// TwinCAT 3 PLC project ProcessControl
// ProgramVersion: 3.1.4023.0
// libraries:
//   CmpBitmapPool, * (System)
//   Tc2_Standard, * (Beckhoff Automation GmbH)
//   Tc2_System, * (Beckhoff Automation GmbH)
//   Tc3_Module, * (Beckhoff Automation GmbH)
//   VisuSymbols,3.5.10.0,System
// project tree:
//   DUTs/ ATV_Status.TcDUT
//   / GlobalTextList.TcGTLO, PlcTask.TcTTO, Visualization Manager.TcVMO (not stored), VISU_TASK.TcTTO
//   GVLs/ drive.TcGVL, Pyrotime.TcGVL, Pyrotime_1.TcGVL
//   POUs/ CabinetSwitch.TcPOU, MAIN.TcPOU, FullProcess.TcPOU, FeedMotor1Manualcontrol.TcPOU, FeedMotor2Manualcontrol.TcPOU, ProcessLamp.TcPOU, RemovalProgram.TcPOU, Scaling.TcPOU, ShortProcess.TcPOU, ValveManualControl.TcPOU
//   VISUs/ ImagePool.TcIPO (not stored), Visualization.TcVIS
// real-time tasks:
//   TASK PlcTask: cycle T#10ms, priority 20, ADS port 350
//   TASK VISU_TASK: cycle T#200000us, priority 30, ADS port 351
// I/O:
//   DEVICE Device 3 (EtherCAT), AmsNetId 5.27.137.92.4.1
//     Box 2 (ATV320 EtherCAT) [ATV320 EtherCAT]
//   DEVICE Device 2 (CX-BK)
//     Box 1 (CX-BK)
// variable links:
//   ProcessControl/ProcessControl Instance <-> Device 2 (CX-BK)/Box 1 (CX-BK)
//     PlcTask Inputs/drive.RawThermoCouple1Value <-> Term 8 (KL3052)/Channel 1/Data In
//     PlcTask Inputs/drive.RawThermoCouple2Value <-> Term 8 (KL3052)/Channel 2/Data In
//     PlcTask Inputs/drive.RemovalSwitch <-> Term 2 (KL1104)/Channel 2/Input
//     PlcTask Inputs/drive.ValveSwitch <-> Term 2 (KL1104)/Channel 3/Input
//     PlcTask Inputs/drive.bEstop <-> Term 2 (KL1104)/Channel 1/Input
//     PlcTask Inputs/drive.bM1switch <-> Term 6 (KL1408)/Channel 2/Input
//     PlcTask Inputs/drive.bM2switch <-> Term 6 (KL1408)/Channel 1/Input
//     PlcTask Inputs/drive.bShortFeed <-> Term 6 (KL1408)/Channel 4/Input
//     PlcTask Inputs/drive.bStartProcess <-> Term 6 (KL1408)/Channel 3/Input
//     PlcTask Outputs/drive.CloseBottomValve <-> Term 3 (KL2114)/Channel 1/Output
//     PlcTask Outputs/drive.CloseTopValve <-> Term 3 (KL2114)/Channel 3/Output
//     PlcTask Outputs/drive.OpenBottomValve <-> Term 3 (KL2114)/Channel 4/Output
//     PlcTask Outputs/drive.OpenTopValve <-> Term 3 (KL2114)/Channel 2/Output
//     PlcTask Outputs/drive.bEmergencyLamp1 <-> Term 7 (KL2408)/Channel 3/Output
//     PlcTask Outputs/drive.bEmptySystemSwitchLamp <-> Term 5 (KL2114)/Channel 4/Output
//     PlcTask Outputs/drive.bFeedMotor2 <-> Term 7 (KL2408)/Channel 6/Output
//     PlcTask Outputs/drive.bM1active <-> Term 4 (KL2114)/Channel 4/Output
//     PlcTask Outputs/drive.bM2active <-> Term 4 (KL2114)/Channel 3/Output
//     PlcTask Outputs/drive.bProcessActive <-> Term 4 (KL2114)/Channel 1/Output
//     PlcTask Outputs/drive.bRemovalMotor <-> Term 5 (KL2114)/Channel 1/Output
//     PlcTask Outputs/drive.bRemovalSequenceLamp <-> Term 5 (KL2114)/Channel 2/Output
//     PlcTask Outputs/drive.bVacuum <-> Term 7 (KL2408)/Channel 5/Output
//     PlcTask Outputs/drive.bValveLamp <-> Term 4 (KL2114)/Channel 2/Output
//     PlcTask Outputs/drive.bValveSwitchLamp <-> Term 5 (KL2114)/Channel 3/Output
//     PlcTask Outputs/drive.bfeedmotorSwitchlamp <-> Term 7 (KL2408)/Channel 2/Output
//     PlcTask Outputs/drive.bremovalmotorSwitchlamp <-> Term 7 (KL2408)/Channel 1/Output
//     PlcTask Outputs/drive.bstartprocessSwitchlamp <-> Term 7 (KL2408)/Channel 4/Output
//   ProcessControl/ProcessControl Instance <-> Device 3 (EtherCAT)/Box 2 (ATV320 EtherCAT)
//     PlcTask Inputs/drive.ATV_TPDO_Input1_Status_Word <-> Inputs/Status word
//     PlcTask Inputs/drive.ATV_TPDO_Input2_Control_Effort <-> Inputs/Control Effort
//     PlcTask Outputs/drive.ATV_RPDO_Output1_Control_Word <-> Outputs/Control word
//     PlcTask Outputs/drive.ATV_RPDO_Output2_Target_Velocity <-> Outputs/Target Velocity

CONFIGURATION ProcessControl
    RESOURCE PLC ON TwinCAT3
        TASK PlcTask(INTERVAL := T#10ms, PRIORITY := 20);
        TASK VISU_TASK(INTERVAL := T#200000us, PRIORITY := 30);
        PROGRAM MAIN WITH PlcTask : MAIN;
        PROGRAM VisuElems_Visu_Prg WITH VISU_TASK : VisuElems.Visu_Prg;
    END_RESOURCE
END_CONFIGURATION

// ---- DUTs/ATV_Status.TcDUT
{attribute 'qualified_only'}
{attribute 'strict'}
TYPE ATV_Status :
(
    SwitchON_disabled := 592, //0
	rdy2SwitchON := 561,	// 6 
	SwitchedON := 563,		// 7 hexadecimal. Motor is in a state, ready to be turned on but not actually on
	OP_Enabled := 1591		//15 hexadecimal. Motor is actually in operation
)   WORD := SwitchON_disabled;
END_TYPE

// ---- GVLs/drive.TcGVL
{attribute 'qualified_only'}
VAR_GLOBAL
	// -------- motor 1 params --------------------------	
	ATV_State AT %I* : WORD;
	PLC_state AT %I* : UINT;
	ATV_TPDO_Input1_Status_Word AT %I* : WORD;
	ATV_TPDO_Input2_Control_Effort AT %I* : WORD;
	ATV_TPDO_Input3 AT %I* : WORD; 
	ATV_TPDO_Input4 AT %I* : WORD;
	ATV_TPDO_Input5 AT %I* : WORD;
	ATV_TPDO_Input6 AT %I* : WORD;
	ATV_RPDO_Output1_Control_Word AT %Q* : WORD;
	ATV_RPDO_Output2_Target_Velocity AT %Q* : WORD;
	ATV_RPDO_Output3 AT %Q* : WORD; 
	ATV_RPDO_Output4 AT %Q* : WORD; 
	ATV_RPDO_Output5 AT %Q* : WORD; 
	ATV_RPDO_Output6 AT %Q* : WORD; 
// -------- motor 1 params --------------------------

// -------- motor 2 params --------------------------
{attribute 'OPC.UA.DA' := '1'} 
bRemovalMotor AT %Q* : BOOL;
// -------- motor 2 params --------------------------

//------------ fan params ----------------
{attribute 'OPC.UA.DA' := '1'} 
bGasfan AT %Q* : BOOL;
//------------- fan params ------------------

//---------- motor 3 params--------------------------
{attribute 'OPC.UA.DA' := '1'} 
bFeedMotor2 AT %Q* : BOOL;
//----------- motor 3 params ------------------------

//---------- switches -------------------------------
{attribute 'OPC.UA.DA' := '1'} 
bStartProcess AT %I* :BOOL;

bEstop      AT %I* 	 :BOOL; 

bM1switch AT %I* 	 :BOOL; 

bM2switch AT %I* 	 :BOOL;

RemovalSwitch AT %I* :BOOL;

{attribute 'OPC.UA.DA' := '1'} 
bShortFeed AT %I* 	 :BOOL; 

bCompressor  	 	 :BOOL; 

{attribute 'OPC.UA.DA' := '1'} 
ValveSwitch AT %I* 	 :BOOL;
//---------- switches -----------------------------

// ---------Lamps----------------------------------
// lamps on the door of the cabinet 
bEmergencyLamp1 AT %Q*   :BOOL; 

{attribute 'OPC.UA.DA' := '1'} 
bProcessActive AT %Q*    :BOOL;
 
bRemovalSequenceLamp AT %Q*   :BOOL;

{attribute 'OPC.UA.DA' := '1'} 
bM1active 		AT %Q* 	 :BOOL;

{attribute 'OPC.UA.DA' := '1'} 
bM2active		AT %Q* 	 :BOOL;

bVacuumActive   AT %Q* 	 :BOOL; 

bValveLamp AT %Q* 		 :BOOL; 

bFeedMotor2Lamp AT %Q*   :BOOL;

//----- lamps inside the switches -------------
bstartprocessSwitchlamp AT %Q* :BOOL;

bfeedmotorSwitchlamp AT %Q* :BOOL; 

bremovalmotorSwitchlamp AT %Q* :BOOL;  

bValveSwitchLamp AT %Q* :BOOL;

bEmptySystemSwitchLamp at %Q* :BOOL; 
// ---------Lamps-----------------------------------

//----------- counter variables ---------------------

ifeedmotor1count: INT;
itopvalvecount: INT := 1;

//----------- counter variables ---------------------


//----status variables-------------
bM1run  	 :BOOL;
ProcessActive :BOOL;
bM1status    : BOOL;    				// tells if the motor is on/off
//-----status variables------------



//---------Valve control ------------------------------------
{attribute 'OPC.UA.DA' := '1'} 
OpenTopValve AT %Q* : BOOL;

{attribute 'OPC.UA.DA' := '1'} 
CloseTopValve AT %Q*: BOOL;
 
{attribute 'OPC.UA.DA' := '1'} 
OpenBottomValve AT %Q* : BOOL;

{attribute 'OPC.UA.DA' := '1'} 
CloseBottomValve AT %Q*: BOOL; 
//----------Valve control -----------------------------------

//----- Vacuum pump --------------------------------------
{attribute 'OPC.UA.DA' := '1'} 
bVacuum  AT %Q*	 : BOOL;
//-----Vacuum pump ---------------------------------------


//------------Temperature variables ---------------------------
RawThermoCouple1Value  AT %I* :INT;
ScaledThermoCouple1Value: REAL; 
RawThermoCouple2Value AT %I*: INT;

{attribute 'OPC.UA.DA' := '1'} 
ScaledThermoCouple2Value: REAL; 
//-----------Temperature variables -----------------------------

END_VAR

// ---- GVLs/Pyrotime.TcGVL
{attribute 'qualified_only'}

// Times used for testing.
VAR_GLOBAL
	tStartDelay: TIME := T#1S;
	tInitFeed: TIME := T#344S; //344s
	tShortFeed: TIME := T#118S; //118s
	tTempFall: TIME:= T#2S;
	tRemovalMotor: TIME := T#114S; //114s
	tValve2: TIME := T#3S;
	tVacuum: TIME := t#10s;
END_VAR

// ---- GVLs/Pyrotime_1.TcGVL
{attribute 'qualified_only'}

// These times are for testing. They are much shorter than the original times
VAR_GLOBAL
	tStartDelay: TIME := T#1S;
	tInitFeed: TIME := T#4S; //344s
	tShortFeed: TIME := T#5S; //118s
	tTempFall: TIME:= T#2S;
	tRemovalMotor: TIME := T#5S; //114s
	tValve2: TIME := T#2S;
END_VAR

// ---- POUs/MAIN.TcPOU
PROGRAM MAIN
VAR
END_VAR

ProcessLamp();
FullProcess();
ShortProcess(); 
FeedMotor1Manualcontrol();
CabinetSwitch();
ValveManualControl();
Scaling();
FeedMotor2Manualcontrol();
RemovalProgram();

END_PROGRAM

// ---- POUs/ProcessLamp.TcPOU
PROGRAM ProcessLamp
VAR
END_VAR

// Written 10.08.2023 by Daniel Kelly

// The purpose of this POU is to provide control to the lamps on the 
// front of the cabinet via their switches

drive.bM1active := drive.bM1switch;
drive.bM2active := drive.bM2switch; 
drive.bProcessActive := drive.bShortFeed OR drive.bStartProcess;
drive.bRemovalSequenceLamp := drive.RemovalSwitch;
drive.bValveLamp := drive.ValveSwitch;

END_PROGRAM

// ---- POUs/FullProcess.TcPOU
PROGRAM FullProcess
VAR
END_VAR
// written 7.08.2023 by Daniel Kelly

// This program is the full version of the process. It includes longer feeding 
// and residence times
// RValveOff turns off the solenoids on the righthandside incase they were already on
// OpenValve opens the top valve
// Step Vacuum removes the excess air from inside the pipe via the vacuum
//waitTemp waits until the temperature is at least 350 degrees celsius
// BiomassFeed operates the second feeding motor
// Init_Feed operates the main feeding motor
// wait600 waits until temperature is 600
// GasFanON turns on the gas fan
// ShortFeed turns on the main feeding motor 1
// ExitMotor turns on the removal motor and opens the top valve
// Valve2Open opens the bottom valve
// Valve2Close closes the bottom valve
// SolenoidsOff turns off the solenoids incase they were on
// AirRemoval removes the air from the pipe
// turnoff1 etc. turns off the devices such as the valves and feeding motor 2

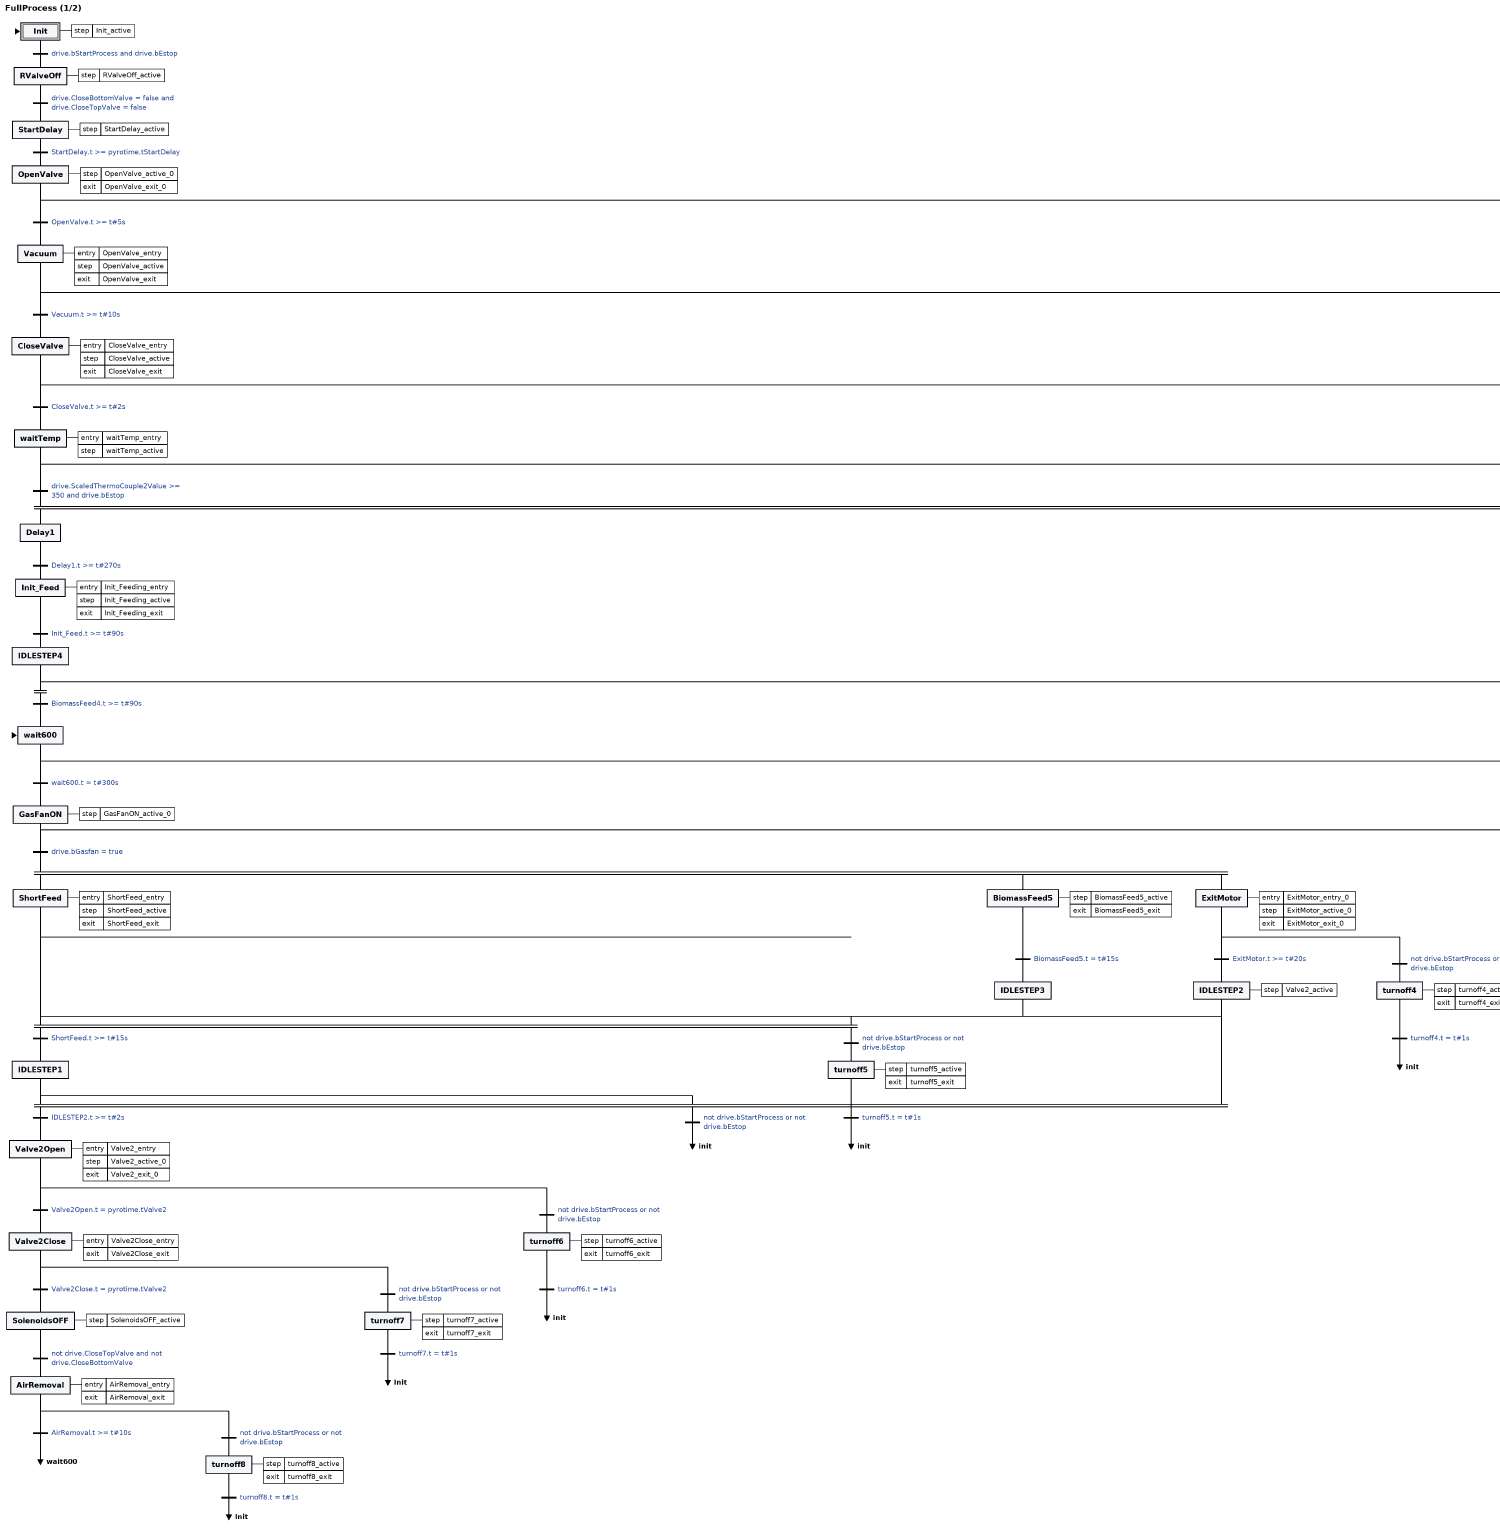
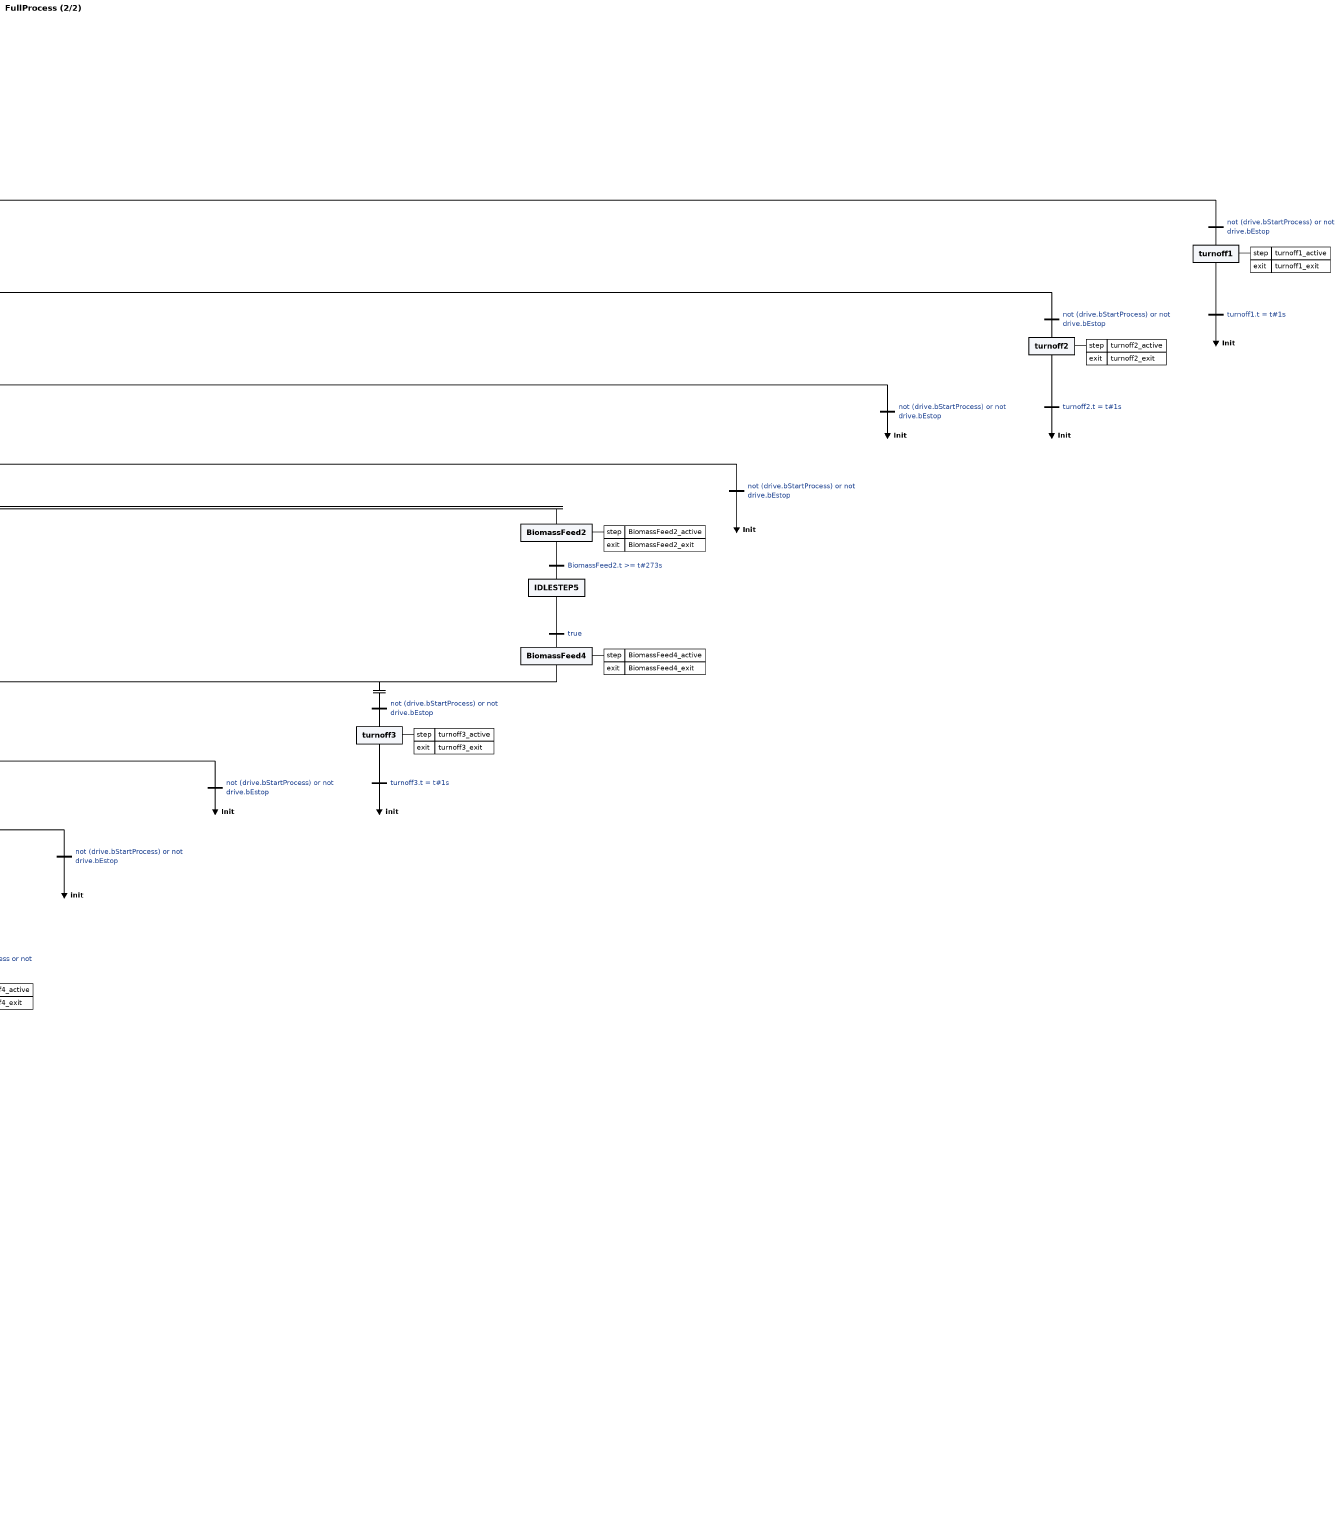
INITIAL_STEP Init:
    Init_active(N);  // step action
END_STEP
TRANSITION FROM Init TO RValveOff
    := drive.bStartProcess and drive.bEstop;
END_TRANSITION
STEP RValveOff:
    RValveOff_active(N);  // step action
END_STEP
TRANSITION FROM RValveOff TO StartDelay
    := drive.CloseBottomValve = false and drive.CloseTopValve = false;
END_TRANSITION
STEP StartDelay:
    StartDelay_active(N);  // step action
END_STEP
TRANSITION FROM StartDelay TO OpenValve
    := StartDelay.t >= pyrotime.tStartDelay;
END_TRANSITION
STEP OpenValve:
    OpenValve_active_0(N);  // step action
    OpenValve_exit_0(P0);  // exit action
END_STEP
TRANSITION FROM OpenValve TO Vacuum
    := OpenValve.t >= t#5s;
END_TRANSITION
TRANSITION FROM OpenValve TO turnoff1
    := not (drive.bStartProcess) or not drive.bEstop;
END_TRANSITION
STEP turnoff1:
    turnoff1_active(N);  // step action
    turnoff1_exit(P0);  // exit action
END_STEP
TRANSITION FROM turnoff1 TO Init
    := turnoff1.t = t#1s;
END_TRANSITION
STEP Vacuum:
    OpenValve_entry(P1);  // entry action
    OpenValve_active(N);  // step action
    OpenValve_exit(P0);  // exit action
END_STEP
TRANSITION FROM Vacuum TO CloseValve
    := Vacuum.t >= t#10s;
END_TRANSITION
TRANSITION FROM Vacuum TO turnoff2
    := not (drive.bStartProcess) or not drive.bEstop;
END_TRANSITION
STEP turnoff2:
    turnoff2_active(N);  // step action
    turnoff2_exit(P0);  // exit action
END_STEP
TRANSITION FROM turnoff2 TO Init
    := turnoff2.t = t#1s;
END_TRANSITION
STEP CloseValve:
    CloseValve_entry(P1);  // entry action
    CloseValve_active(N);  // step action
    CloseValve_exit(P0);  // exit action
END_STEP
TRANSITION FROM CloseValve TO waitTemp
    := CloseValve.t >= t#2s;
END_TRANSITION
TRANSITION FROM CloseValve TO Init
    := not (drive.bStartProcess) or not drive.bEstop;
END_TRANSITION
STEP waitTemp:
    waitTemp_entry(P1);  // entry action
    waitTemp_active(N);  // step action
END_STEP
TRANSITION FROM waitTemp TO (Delay1, BiomassFeed2)
    := drive.ScaledThermoCouple2Value >= 350 and drive.bEstop;
END_TRANSITION
TRANSITION FROM waitTemp TO Init
    := not (drive.bStartProcess) or not drive.bEstop;
END_TRANSITION
STEP Delay1:
END_STEP
TRANSITION FROM Delay1 TO Init_Feed
    := Delay1.t >= t#270s;
END_TRANSITION
STEP Init_Feed:
    Init_Feeding_entry(P1);  // entry action
    Init_Feeding_active(N);  // step action
    Init_Feeding_exit(P0);  // exit action
END_STEP
TRANSITION FROM Init_Feed TO IDLESTEP4
    := Init_Feed.t >= t#90s;
END_TRANSITION
STEP IDLESTEP4:
END_STEP
STEP BiomassFeed2:
    BiomassFeed2_active(N);  // step action
    BiomassFeed2_exit(P0);  // exit action
END_STEP
TRANSITION FROM BiomassFeed2 TO IDLESTEP5
    := BiomassFeed2.t >= t#273s;
END_TRANSITION
STEP IDLESTEP5:
END_STEP
TRANSITION FROM IDLESTEP5 TO BiomassFeed4
    := true;
END_TRANSITION
STEP BiomassFeed4:
    BiomassFeed4_active(N);  // step action
    BiomassFeed4_exit(P0);  // exit action
END_STEP
TRANSITION FROM (IDLESTEP4, BiomassFeed4) TO wait600
    := BiomassFeed4.t >= t#90s;
END_TRANSITION
TRANSITION FROM (IDLESTEP4, BiomassFeed4) TO turnoff3
    := not (drive.bStartProcess) or not drive.bEstop;
END_TRANSITION
STEP turnoff3:
    turnoff3_active(N);  // step action
    turnoff3_exit(P0);  // exit action
END_STEP
TRANSITION FROM turnoff3 TO init
    := turnoff3.t = t#1s;
END_TRANSITION
STEP wait600:
END_STEP
TRANSITION FROM wait600 TO GasFanON
    := wait600.t = t#300s;
END_TRANSITION
STEP GasFanON:
    GasFanON_active_0(N);  // step action
END_STEP
TRANSITION FROM GasFanON TO (ShortFeed, BiomassFeed5, ExitMotor)
    := drive.bGasfan = true;
END_TRANSITION
TRANSITION FROM GasFanON TO init
    := not (drive.bStartProcess) or not drive.bEstop;
END_TRANSITION
TRANSITION FROM wait600 TO Init
    := not (drive.bStartProcess) or not drive.bEstop;
END_TRANSITION
STEP ShortFeed:
    ShortFeed_entry(P1);  // entry action
    ShortFeed_active(N);  // step action
    ShortFeed_exit(P0);  // exit action
END_STEP
STEP BiomassFeed5:
    BiomassFeed5_active(N);  // step action
    BiomassFeed5_exit(P0);  // exit action
END_STEP
TRANSITION FROM BiomassFeed5 TO IDLESTEP3
    := BiomassFeed5.t = t#15s;
END_TRANSITION
STEP IDLESTEP3:
END_STEP
TRANSITION FROM (ShortFeed, IDLESTEP3) TO IDLESTEP1
    := ShortFeed.t >= t#15s;
END_TRANSITION
TRANSITION FROM (ShortFeed, IDLESTEP3) TO turnoff5
    := not drive.bStartProcess or not drive.bEstop;
END_TRANSITION
STEP turnoff5:
    turnoff5_active(N);  // step action
    turnoff5_exit(P0);  // exit action
END_STEP
TRANSITION FROM turnoff5 TO init
    := turnoff5.t = t#1s;
END_TRANSITION
STEP IDLESTEP1:
END_STEP
STEP ExitMotor:
    ExitMotor_entry_0(P1);  // entry action
    ExitMotor_active_0(N);  // step action
    ExitMotor_exit_0(P0);  // exit action
END_STEP
TRANSITION FROM ExitMotor TO IDLESTEP2
    := ExitMotor.t >= t#20s;
END_TRANSITION
TRANSITION FROM ExitMotor TO turnoff4
    := not drive.bStartProcess or not drive.bEstop;
END_TRANSITION
STEP turnoff4:
    turnoff4_active(N);  // step action
    turnoff4_exit(P0);  // exit action
END_STEP
TRANSITION FROM turnoff4 TO init
    := turnoff4.t = t#1s;
END_TRANSITION
STEP IDLESTEP2:
    Valve2_active(N);  // step action
END_STEP
TRANSITION FROM (IDLESTEP1, IDLESTEP2) TO Valve2Open
    := IDLESTEP2.t >= t#2s;
END_TRANSITION
TRANSITION FROM (IDLESTEP1, IDLESTEP2) TO init
    := not drive.bStartProcess or not drive.bEstop;
END_TRANSITION
STEP Valve2Open:
    Valve2_entry(P1);  // entry action
    Valve2_active_0(N);  // step action
    Valve2_exit_0(P0);  // exit action
END_STEP
TRANSITION FROM Valve2Open TO Valve2Close
    := Valve2Open.t = pyrotime.tValve2;
END_TRANSITION
TRANSITION FROM Valve2Open TO turnoff6
    := not drive.bStartProcess or not drive.bEstop;
END_TRANSITION
STEP turnoff6:
    turnoff6_active(N);  // step action
    turnoff6_exit(P0);  // exit action
END_STEP
TRANSITION FROM turnoff6 TO init
    := turnoff6.t = t#1s;
END_TRANSITION
STEP Valve2Close:
    Valve2Close_entry(P1);  // entry action
    Valve2Close_exit(P0);  // exit action
END_STEP
TRANSITION FROM Valve2Close TO SolenoidsOFF
    := Valve2Close.t = pyrotime.tValve2;
END_TRANSITION
TRANSITION FROM Valve2Close TO turnoff7
    := not drive.bStartProcess or not drive.bEstop;
END_TRANSITION
STEP turnoff7:
    turnoff7_active(N);  // step action
    turnoff7_exit(P0);  // exit action
END_STEP
TRANSITION FROM turnoff7 TO Init
    := turnoff7.t = t#1s;
END_TRANSITION
STEP SolenoidsOFF:
    SolenoidsOFF_active(N);  // step action
END_STEP
TRANSITION FROM SolenoidsOFF TO AirRemoval
    := not drive.CloseTopValve and not drive.CloseBottomValve;
END_TRANSITION
STEP AirRemoval:
    AirRemoval_entry(P1);  // entry action
    AirRemoval_exit(P0);  // exit action
END_STEP
TRANSITION FROM AirRemoval TO wait600
    := AirRemoval.t >= t#10s;
END_TRANSITION
TRANSITION FROM AirRemoval TO turnoff8
    := not drive.bStartProcess or not drive.bEstop;
END_TRANSITION
STEP turnoff8:
    turnoff8_active(N);  // step action
    turnoff8_exit(P0);  // exit action
END_STEP
TRANSITION FROM turnoff8 TO Init
    := turnoff8.t = t#1s;
END_TRANSITION

ACTION AirRemoval_entry:
drive.bVacuum := TRUE;
END_ACTION

ACTION AirRemoval_exit:
drive.bVacuum := FALSE;
END_ACTION

ACTION BiomassFeed_active:
drive.bFeedMotor2 := true;
END_ACTION

ACTION BiomassFeed_exit:
drive.bFeedMotor2 := false;
END_ACTION

ACTION BiomassFeed2_active:
drive.bFeedMotor2 := TRUE;
END_ACTION

ACTION BiomassFeed2_exit:
drive.bFeedMotor2 := FALSE;
END_ACTION

ACTION BiomassFeed4_active:
drive.bFeedMotor2 := TRUE;
END_ACTION

ACTION BiomassFeed4_exit:
drive.bFeedMotor2 := false;
END_ACTION

ACTION BiomassFeed5_active:
drive.bFeedMotor2 := true;
END_ACTION

ACTION BiomassFeed5_exit:
drive.bFeedMotor2 := false;
END_ACTION

ACTION CloseValve_active:
drive.CloseTopValve := TRUE;
drive.CloseBottomValve := FALSE;
END_ACTION

ACTION CloseValve_entry:
//drive.RightSolenoid := TRUE;
END_ACTION

ACTION CloseValve_exit:
drive.CloseTopValve := FALSE;
END_ACTION

ACTION ExitMotor_active_0:
drive.bRemovalMotor := TRUE;
drive.bM2active := TRUE; // lamp variable



drive.OpenTopValve := TRUE; // opens valve
drive.CloseTopValve := FALSE;
END_ACTION

ACTION ExitMotor_entry_0:

END_ACTION

ACTION ExitMotor_exit_0:
 
drive.CloseTopValve := TRUE; //closes valve
drive.OpenTopValve := FALSE;

drive.bM2active := FALSE; // lamp variable ; turns lamp off
drive.bRemovalMotor := FALSE; // turns the removal motor off
END_ACTION

ACTION ExitMotor1_active:
drive.bRemovalMotor := TRUE;
END_ACTION

ACTION GasFanOFF_active:
drive.bGasfan := false;
END_ACTION

ACTION GasFanOFF_active_0:
drive.bGasfan := false;
END_ACTION

ACTION GasFanOn_active:
drive.bGasfan := TRUE;
END_ACTION

ACTION GasFanON_active_0:
drive.bGasfan := TRUE;
END_ACTION

ACTION Init_active:
//drive.ATV_RPDO_Output1_Control_Word := 0;
//drive.bRemovalMotor := FALSE; 
//drive.bProcessActive := FALSE;
//drive.LeftSolenoid := FALSE;
//drive.LeftSolenoid2 := FALSE; 
//drive.RightSolenoid := TRUE;
//drive.RightSolenoid2 := TRUE;
 
drive.ifeedmotor1count := 0;
END_ACTION

ACTION Init_Feeding_active:
IF drive.ATV_TPDO_Input1_Status_Word = ATV_Status.rdy2SwitchON THEN 
	drive.ATV_RPDO_Output1_Control_Word := 7; //SwitchedON
END_IF

IF drive.ATV_TPDO_Input1_Status_Word = ATV_Status.SwitchedON THEN 
	drive.ATV_RPDO_Output1_Control_Word := 15; //OP_Enabled
	drive.bM1active := TRUE; // lamp goes on
	drive.bM1status := TRUE;  // status variable
END_IF
END_ACTION

ACTION Init_Feeding_entry:
drive.ATV_RPDO_Output1_Control_Word := 6; //rdy2SwitchON
drive.ATV_RPDO_Output2_Target_Velocity := 1000;
END_ACTION

ACTION Init_Feeding_exit:


IF drive.bM1status = TRUE THEN 
	drive.ifeedmotor1count := drive.ifeedmotor1count + 1;
END_IF

drive.ATV_RPDO_Output1_Control_Word := 7; //switchedON, ready mode
drive.bM1active := FALSE;  // lamp off
drive.bM1status := FALSE;  // status variable for feeding motor 1
END_ACTION

ACTION OpenValve_active:

END_ACTION

ACTION OpenValve_active_0:
drive.OpenTopValve := TRUE;
drive.CloseTopValve := FALSE;
END_ACTION

ACTION OpenValve_entry:

drive.bVacuum := TRUE;
END_ACTION

ACTION OpenValve_exit:
drive.bVacuum := FALSE;
END_ACTION

ACTION OpenValve_exit_0:
drive.OpenTopValve := false;
END_ACTION

ACTION ProcessActive_active:
IF drive.bStartProcess THEN 
	drive.bProcessActive := TRUE;
ELSE 
	drive.bProcessActive := FALSE; 
END_IF
END_ACTION

ACTION RValveOff_active:
drive.CloseTopValve := FALSE;
drive.CloseBottomValve := FALSE;
END_ACTION

ACTION ShortFeed_active:
IF drive.ATV_TPDO_Input1_Status_Word = ATV_Status.rdy2SwitchON THEN 
	drive.ATV_RPDO_Output1_Control_Word := 7;
END_IF

IF drive.ATV_TPDO_Input1_Status_Word = ATV_Status.SwitchedON THEN
			drive.bM1run := TRUE; //counter variable
			drive.bM1active := TRUE;
			drive.ATV_RPDO_Output1_Control_Word := 15;
END_IF
END_ACTION

ACTION ShortFeed_entry:
drive.ATV_RPDO_Output2_Target_Velocity := 1000;
drive.ATV_RPDO_Output1_Control_Word := 6;
END_ACTION

ACTION ShortFeed_exit:


drive.bM1run := FALSE;
drive.bM1active := FALSE; 
drive.ATV_RPDO_Output1_Control_Word := 7;
END_ACTION

ACTION SolenoidsOFF_active:
drive.CloseTopValve := FALSE;
drive.CloseBottomValve := FALSE;
END_ACTION

ACTION StartDelay_active:
IF drive.bStartProcess THEN 
	drive.bProcessActive := TRUE;
ELSE 
	drive.bProcessActive := FALSE; 
END_IF
END_ACTION

ACTION turnoff1_active:
drive.CloseTopValve := TRUE;
drive.OpenTopValve := FALSE;
END_ACTION

ACTION turnoff1_exit:
drive.CloseTopValve := FALSE;
END_ACTION

ACTION turnoff2_active:
drive.bVacuum := FALSE;
END_ACTION

ACTION turnoff2_exit:

END_ACTION

ACTION turnoff3_active:
drive.bM1status := FALSE;
drive.bFeedMotor2 := FALSE;
drive.bM1active := FALSE;
END_ACTION

ACTION turnoff3_exit:

END_ACTION

ACTION turnoff4_active:
drive.bRemovalMotor := FALSE;
drive.bM2active := FALSE;

drive.OpenTopValve := FALSE;
drive.CloseTopValve := TRUE;
END_ACTION

ACTION turnoff4_exit:
drive.CloseTopValve := false;
END_ACTION

ACTION turnoff5_active:
drive.bFeedMotor2 := FALSE;


drive.bRemovalMotor := FALSE;
drive.bM2active := FALSE;

drive.OpenTopValve := FALSE;
drive.CloseTopValve := TRUE;
END_ACTION

ACTION turnoff5_exit:

END_ACTION

ACTION turnoff6_active:
drive.CloseBottomValve := TRUE;
drive.OpenBottomValve := FALSE;
END_ACTION

ACTION turnoff6_exit:
drive.CloseBottomValve := FALSE;
END_ACTION

ACTION turnoff7_active:
drive.CloseBottomValve := TRUE;
END_ACTION

ACTION turnoff7_exit:
drive.CloseBottomValve := FALSE;
END_ACTION

ACTION turnoff8_active:
drive.bVacuum := false;
END_ACTION

ACTION turnoff8_exit:

END_ACTION

ACTION Vacuum_entry:

END_ACTION

ACTION Vacuum_exit:
drive.bVacuum := FALSE;
END_ACTION

ACTION Valve2_active:

END_ACTION

ACTION Valve2_active_0:

END_ACTION

ACTION Valve2_entry:
drive.OpenBottomValve := TRUE;
END_ACTION

ACTION Valve2_exit_0:
drive.OpenBottomValve := FALSE;
END_ACTION

ACTION Valve2Close_entry:
drive.CloseBottomValve := TRUE;
END_ACTION

ACTION Valve2Close_exit:
 drive.CloseBottomValve := FALSE;
END_ACTION

ACTION waitTemp_active:

END_ACTION

ACTION waitTemp_entry:

END_ACTION

END_PROGRAM

// ---- POUs/ShortProcess.TcPOU
	PROGRAM ShortProcess
VAR
	cM1startCount : INT;
	
END_VAR
// written 7.08.2023 by Daniel Kelly

// Program is a shorter version of the full process cycle

//Step RValveOff turns off the top and bottom closing valves
// Step Wait500 waits until the temperature is at 500
//Step GasFanOn turns on the gas fan
// Step waittemp is the residence time
//Step ShortFeed and Biomass Feed run simultaneously to feed the biomass into the furnace
// Step ExitMotor operates the removal motor and opens the top valve
// Steps M1override and M2override overrides the original motor operating time.
//Step Valve2Open opens the bottom valve
// Step Valve2Close closes the bottom valve

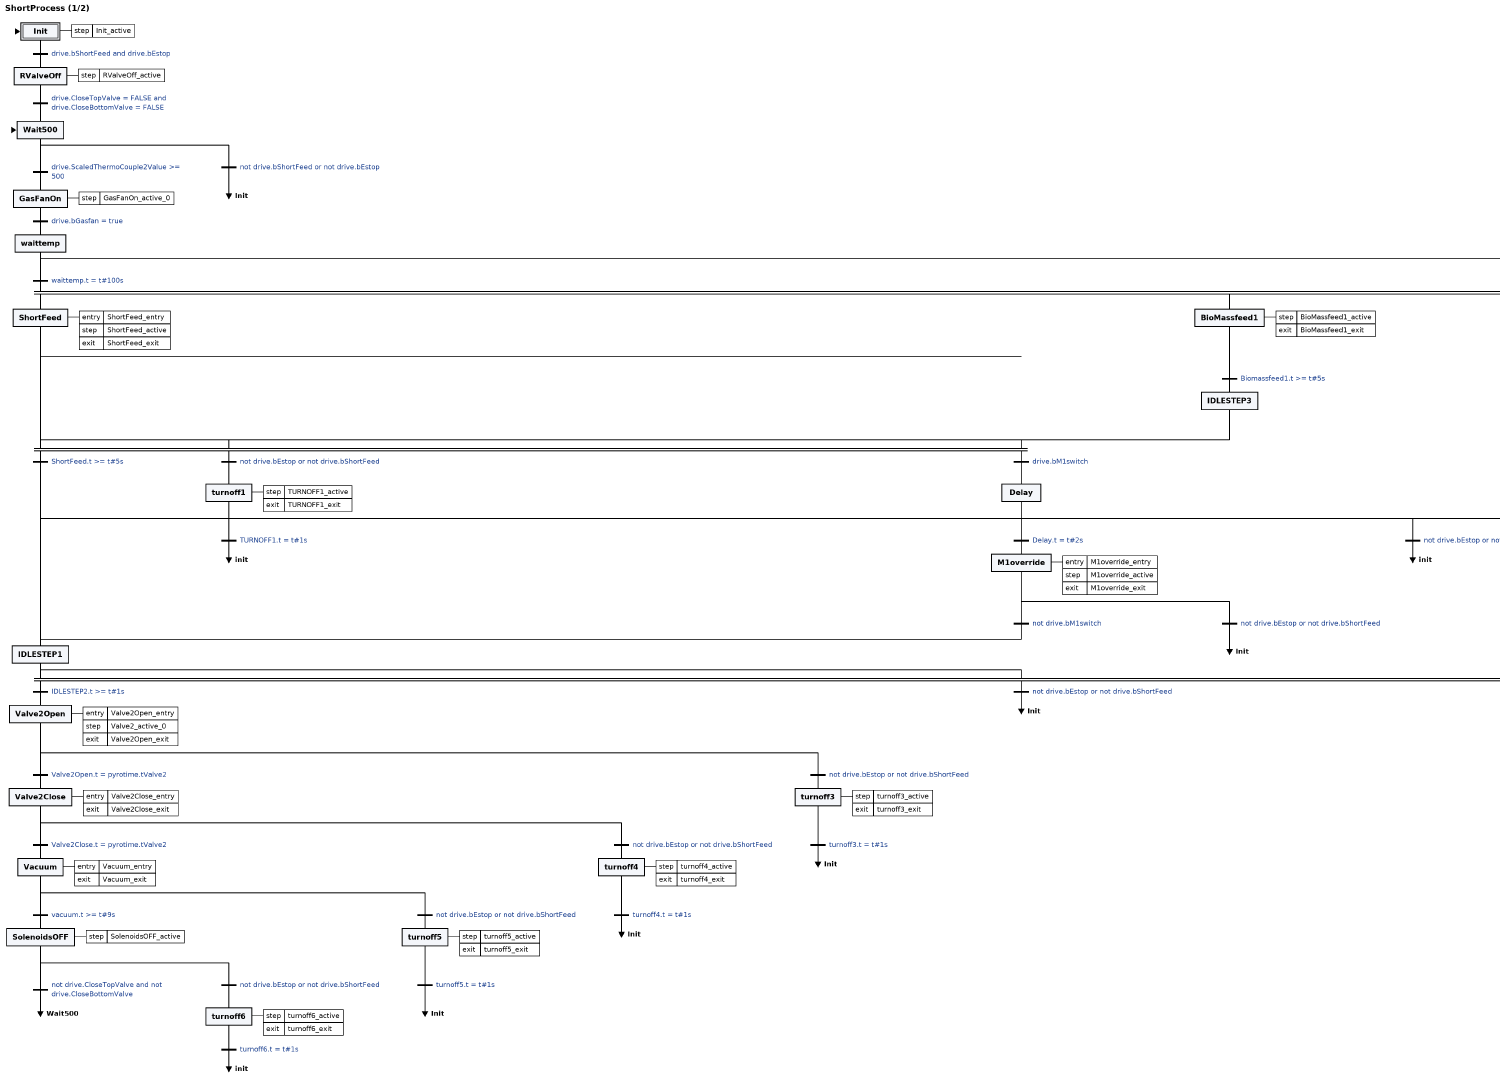
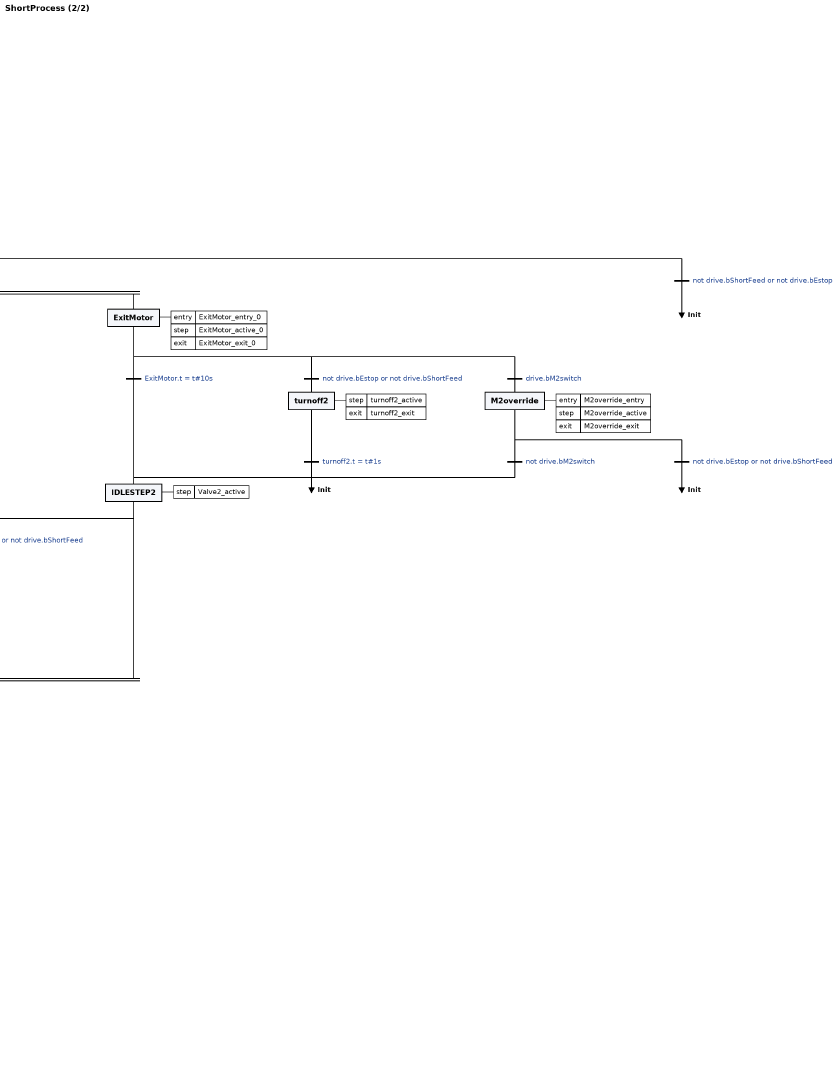
INITIAL_STEP Init:
    Init_active(N);  // step action
END_STEP
TRANSITION FROM Init TO RValveOff
    := drive.bShortFeed and drive.bEstop;
END_TRANSITION
STEP RValveOff:
    RValveOff_active(N);  // step action
END_STEP
TRANSITION FROM RValveOff TO Wait500
    := drive.CloseTopValve = FALSE and drive.CloseBottomValve = FALSE;
END_TRANSITION
STEP Wait500:
END_STEP
TRANSITION FROM Wait500 TO GasFanOn
    := drive.ScaledThermoCouple2Value >= 500;
END_TRANSITION
STEP GasFanOn:
    GasFanOn_active_0(N);  // step action
END_STEP
TRANSITION FROM GasFanOn TO waittemp
    := drive.bGasfan = true;
END_TRANSITION
TRANSITION FROM Wait500 TO Init
    := not drive.bShortFeed or not drive.bEstop;
END_TRANSITION
STEP waittemp:
END_STEP
TRANSITION FROM waittemp TO (ShortFeed, BioMassfeed1, ExitMotor)
    := waittemp.t = t#100s;
END_TRANSITION
TRANSITION FROM waittemp TO Init
    := not drive.bShortFeed or not drive.bEstop;
END_TRANSITION
STEP ShortFeed:
    ShortFeed_entry(P1);  // entry action
    ShortFeed_active(N);  // step action
    ShortFeed_exit(P0);  // exit action
END_STEP
STEP BioMassfeed1:
    BioMassfeed1_active(N);  // step action
    BioMassfeed1_exit(P0);  // exit action
END_STEP
TRANSITION FROM BioMassfeed1 TO IDLESTEP3
    := Biomassfeed1.t >= t#5s;
END_TRANSITION
STEP IDLESTEP3:
END_STEP
TRANSITION FROM (ShortFeed, IDLESTEP3) TO IDLESTEP1
    := ShortFeed.t >= t#5s;
END_TRANSITION
TRANSITION FROM (ShortFeed, IDLESTEP3) TO turnoff1
    := not drive.bEstop or not drive.bShortFeed;
END_TRANSITION
STEP turnoff1:
    TURNOFF1_active(N);  // step action
    TURNOFF1_exit(P0);  // exit action
END_STEP
TRANSITION FROM turnoff1 TO init
    := TURNOFF1.t = t#1s;
END_TRANSITION
TRANSITION FROM (ShortFeed, IDLESTEP3) TO Delay
    := drive.bM1switch;
END_TRANSITION
STEP Delay:
END_STEP
TRANSITION FROM Delay TO M1override
    := Delay.t = t#2s;
END_TRANSITION
TRANSITION FROM Delay TO init
    := not drive.bEstop or not drive.bShortFeed;
END_TRANSITION
STEP M1override:
    M1override_entry(P1);  // entry action
    M1override_active(N);  // step action
    M1override_exit(P0);  // exit action
END_STEP
TRANSITION FROM M1override TO IDLESTEP1
    := not drive.bM1switch;
END_TRANSITION
TRANSITION FROM M1override TO Init
    := not drive.bEstop or not drive.bShortFeed;
END_TRANSITION
STEP IDLESTEP1:
END_STEP
STEP ExitMotor:
    ExitMotor_entry_0(P1);  // entry action
    ExitMotor_active_0(N);  // step action
    ExitMotor_exit_0(P0);  // exit action
END_STEP
TRANSITION FROM ExitMotor TO IDLESTEP2
    := ExitMotor.t = t#10s;
END_TRANSITION
TRANSITION FROM ExitMotor TO turnoff2
    := not drive.bEstop or not drive.bShortFeed;
END_TRANSITION
STEP turnoff2:
    turnoff2_active(N);  // step action
    turnoff2_exit(P0);  // exit action
END_STEP
TRANSITION FROM turnoff2 TO Init
    := turnoff2.t = t#1s;
END_TRANSITION
TRANSITION FROM ExitMotor TO M2override
    := drive.bM2switch;
END_TRANSITION
STEP M2override:
    M2override_entry(P1);  // entry action
    M2override_active(N);  // step action
    M2override_exit(P0);  // exit action
END_STEP
TRANSITION FROM M2override TO IDLESTEP2
    := not drive.bM2switch;
END_TRANSITION
TRANSITION FROM M2override TO Init
    := not drive.bEstop or not drive.bShortFeed;
END_TRANSITION
STEP IDLESTEP2:
    Valve2_active(N);  // step action
END_STEP
TRANSITION FROM (IDLESTEP1, IDLESTEP2) TO Valve2Open
    := IDLESTEP2.t >= t#1s;
END_TRANSITION
TRANSITION FROM (IDLESTEP1, IDLESTEP2) TO Init
    := not drive.bEstop or not drive.bShortFeed;
END_TRANSITION
STEP Valve2Open:
    Valve2Open_entry(P1);  // entry action
    Valve2_active_0(N);  // step action
    Valve2Open_exit(P0);  // exit action
END_STEP
TRANSITION FROM Valve2Open TO Valve2Close
    := Valve2Open.t = pyrotime.tValve2;
END_TRANSITION
TRANSITION FROM Valve2Open TO turnoff3
    := not drive.bEstop or not drive.bShortFeed;
END_TRANSITION
STEP turnoff3:
    turnoff3_active(N);  // step action
    turnoff3_exit(P0);  // exit action
END_STEP
TRANSITION FROM turnoff3 TO Init
    := turnoff3.t = t#1s;
END_TRANSITION
STEP Valve2Close:
    Valve2Close_entry(P1);  // entry action
    Valve2Close_exit(P0);  // exit action
END_STEP
TRANSITION FROM Valve2Close TO Vacuum
    := Valve2Close.t = pyrotime.tValve2;
END_TRANSITION
TRANSITION FROM Valve2Close TO turnoff4
    := not drive.bEstop or not drive.bShortFeed;
END_TRANSITION
STEP turnoff4:
    turnoff4_active(N);  // step action
    turnoff4_exit(P0);  // exit action
END_STEP
TRANSITION FROM turnoff4 TO Init
    := turnoff4.t = t#1s;
END_TRANSITION
STEP Vacuum:
    Vacuum_entry(P1);  // entry action
    Vacuum_exit(P0);  // exit action
END_STEP
TRANSITION FROM Vacuum TO SolenoidsOFF
    := vacuum.t >= t#9s;
END_TRANSITION
TRANSITION FROM Vacuum TO turnoff5
    := not drive.bEstop or not drive.bShortFeed;
END_TRANSITION
STEP turnoff5:
    turnoff5_active(N);  // step action
    turnoff5_exit(P0);  // exit action
END_STEP
TRANSITION FROM turnoff5 TO Init
    := turnoff5.t = t#1s;
END_TRANSITION
STEP SolenoidsOFF:
    SolenoidsOFF_active(N);  // step action
END_STEP
TRANSITION FROM SolenoidsOFF TO Wait500
    := not drive.CloseTopValve and not drive.CloseBottomValve;
END_TRANSITION
TRANSITION FROM SolenoidsOFF TO turnoff6
    := not drive.bEstop or not drive.bShortFeed;
END_TRANSITION
STEP turnoff6:
    turnoff6_active(N);  // step action
    turnoff6_exit(P0);  // exit action
END_STEP
TRANSITION FROM turnoff6 TO init
    := turnoff6.t = t#1s;
END_TRANSITION

ACTION BioMassfeed1_active:
drive.bFeedMotor2 := TRUE;
drive.bFeedMotor2Lamp := TRUE;
END_ACTION

ACTION BioMassfeed1_exit:
drive.bFeedMotor2 := FALSE;
drive.bFeedMotor2Lamp := FALSE;
END_ACTION

ACTION ExitMotor_active_0:
drive.bRemovalMotor := TRUE; 
drive.bM2active := TRUE; // turns on the lamp

drive.bValveLamp := TRUE; // turns on the valve lamp
drive.OpenTopValve := TRUE; 
drive.CloseTopValve := FALSE;
END_ACTION

ACTION ExitMotor_entry_0:

END_ACTION

ACTION ExitMotor_exit_0:

IF drive.OpenTopValve THEN 
	drive.itopvalvecount := drive.itopvalvecount + 1;
END_IF



drive.CloseTopValve := TRUE;
drive.OpenTopValve := FALSE;



drive.bM2active := FALSE; // lamp off
drive.bRemovalMotor := FALSE;
END_ACTION

ACTION ExitMotor1_active:
drive.bRemovalMotor := TRUE;
END_ACTION

ACTION GasFanOFF_active:
drive.bGasfan := FALSE;
END_ACTION

ACTION GasFanOn_active:
drive.bGasfan := true;
END_ACTION

ACTION GasFanOn_active_0:
drive.bGasfan := true;
END_ACTION

ACTION Init_active:
//drive.ATV_RPDO_Output1_Control_Word := 0;
//drive.bRemovalMotor := FALSE;
//drive.bProcessActive := FALSE; 
//drive.LeftSolenoid := FALSE;
//drive.LeftSolenoid2 := FALSE; 
//drive.RightSolenoid := TRUE;
//drive.RightSolenoid2 := TRUE;

drive.bGasfan := FALSE;
END_ACTION

ACTION Init_Feeding_active:
IF drive.ATV_TPDO_Input1_Status_Word = ATV_Status.rdy2SwitchON THEN 
	drive.ATV_RPDO_Output1_Control_Word := 7; //SwitchedON
END_IF

IF drive.ATV_TPDO_Input1_Status_Word = ATV_Status.SwitchedON THEN 
	drive.ATV_RPDO_Output1_Control_Word := 15; //OP_Enabled
END_IF
END_ACTION

ACTION Init_Feeding_entry:
drive.ATV_RPDO_Output1_Control_Word := 6; //rdy2SwitchON
drive.ATV_RPDO_Output2_Target_Velocity := 1000;
END_ACTION

ACTION Init_Feeding_exit:
drive.ATV_RPDO_Output1_Control_Word := 7; //switchedON
END_ACTION

ACTION M1override_active:
IF drive.ATV_TPDO_Input1_Status_Word = atv_status.rdy2SwitchON THEN 
	drive.ATV_RPDO_Output1_Control_Word := 7;
END_IF

IF drive.ATV_TPDO_Input1_Status_Word = atv_status.SwitchedON THEN 
	drive.ATV_RPDO_Output1_Control_Word := 15;
	drive.bM1active := TRUE; 
END_IF
END_ACTION

ACTION M1override_entry:
drive.ATV_RPDO_Output2_Target_Velocity := 1000;
drive.ATV_RPDO_Output1_Control_Word := 6;
END_ACTION

ACTION M1override_exit:
drive.ATV_RPDO_Output1_Control_Word := 7; 
drive.bM1active := false;
END_ACTION

ACTION M2override_active:

END_ACTION

ACTION M2override_entry:
drive.bRemovalMotor := TRUE; 
drive.bM2active := TRUE;
END_ACTION

ACTION M2override_exit:
drive.bRemovalMotor := FALSE; 
drive.bM2active := FALSE;
END_ACTION

ACTION ProcessACTIVE_active:
drive.bProcessActive := TRUE;
END_ACTION

ACTION RValveOff_active:
drive.CloseTopValve := FALSE;
drive.CloseBottomValve := FALSE;
END_ACTION

ACTION ShortFeed_active:
drive.bRemovalMotor := TRUE;
drive.bM1active := TRUE;

IF drive.ATV_TPDO_Input1_Status_Word = ATV_Status.rdy2SwitchON THEN 
	drive.ATV_RPDO_Output1_Control_Word := 7;
END_IF

IF drive.ATV_TPDO_Input1_Status_Word = ATV_Status.SwitchedON THEN
			drive.bM1run := TRUE; 
			drive.ATV_RPDO_Output1_Control_Word := 15;
END_IF
END_ACTION

ACTION ShortFeed_entry:
drive.ATV_RPDO_Output2_Target_Velocity := 1000;
drive.ATV_RPDO_Output1_Control_Word := 6;
END_ACTION

ACTION ShortFeed_exit:
IF drive.bM1run = TRUE THEN 
	cM1startCount := cM1startCount + 1;
END_IF

drive.bM1run := FALSE;
drive.bM1active := FALSE; 
drive.ATV_RPDO_Output1_Control_Word := 7;
END_ACTION

ACTION SolenoidsOFF_active:
drive.CloseTopValve := FALSE;
drive.CloseBottomValve := FALSE;
END_ACTION

ACTION TURNOFF1_active:
drive.bRemovalMotor := FALSE;
drive.OpenTopValve := FALSE;
drive.CloseTopValve := TRUE;
drive.bM1active := false;
END_ACTION

ACTION TURNOFF1_exit:
drive.CloseBottomValve := FALSE;
drive.CloseTopValve := FALSE;
END_ACTION

ACTION turnoff2_active:
drive.bRemovalMotor := FALSE;
drive.OpenTopValve := FALSE;
drive.CloseTopValve := TRUE;
END_ACTION

ACTION turnoff2_exit:
drive.CloseBottomValve := FALSE;
drive.CloseTopValve := FALSE;
END_ACTION

ACTION turnoff3_active:
drive.bRemovalMotor := FALSE;
drive.OpenTopValve := FALSE;
drive.CloseTopValve := TRUE;
drive.OpenBottomValve := FALSE;
drive.CloseBottomValve := TRUE;
END_ACTION

ACTION turnoff3_exit:
drive.CloseBottomValve := FALSE;
drive.CloseTopValve := FALSE;
END_ACTION

ACTION turnoff4_active:
drive.bRemovalMotor := FALSE;
drive.OpenTopValve := FALSE;
drive.CloseTopValve := TRUE;
drive.OpenBottomValve := FALSE;
drive.CloseBottomValve := TRUE;
END_ACTION

ACTION turnoff4_exit:
drive.CloseBottomValve := FALSE;
drive.CloseTopValve := FALSE;
END_ACTION

ACTION turnoff5_active:
drive.bRemovalMotor := FALSE;
drive.OpenTopValve := FALSE;
drive.CloseTopValve := TRUE;
drive.OpenBottomValve := FALSE;
drive.CloseBottomValve := TRUE;
END_ACTION

ACTION turnoff5_exit:
drive.CloseBottomValve := FALSE;
drive.CloseTopValve := FALSE;
END_ACTION

ACTION turnoff6_active:
drive.bRemovalMotor := FALSE;
drive.OpenTopValve := FALSE;
drive.CloseTopValve := TRUE;
drive.OpenBottomValve := FALSE;
drive.CloseBottomValve := TRUE;
END_ACTION

ACTION turnoff6_exit:
drive.CloseBottomValve := FALSE;
drive.CloseTopValve := FALSE;
END_ACTION

ACTION Vacuum_entry:
IF drive.itopvalvecount >= 5 THEN 
	drive.bVacuum := TRUE; 
END_IF
END_ACTION

ACTION Vacuum_exit:
drive.bVacuum := FALSE;
END_ACTION

ACTION Valve2_active:

END_ACTION

ACTION Valve2_active_0:

END_ACTION

ACTION Valve2_exit:

END_ACTION

ACTION Valve2Close_entry:
drive.CloseBottomValve := TRUE;
END_ACTION

ACTION Valve2Close_exit:
drive.CloseBottomValve := FALSE;
drive.bValveLamp := FALSE;
END_ACTION

ACTION Valve2Open_entry:

IF drive.itopvalvecount >= 5 THEN // Bottom valve opens after top valve has opened 5 times or more
	drive.OpenBottomValve := TRUE;
END_IF
END_ACTION

ACTION Valve2Open_exit:

IF drive.OpenBottomValve THEN  //  counter will reset after bottom valve opens
	drive.itopvalvecount := 1; 
END_IF

drive.OpenBottomValve := FALSE;
END_ACTION

END_PROGRAM

// ---- POUs/FeedMotor1Manualcontrol.TcPOU
PROGRAM FeedMotor1Manualcontrol
VAR
END_VAR
// Written 10.08.2023 by Daniel Kelly

// Program provides manual control of the motor M1 via its switch

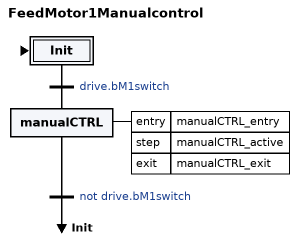
INITIAL_STEP Init:
END_STEP
TRANSITION FROM Init TO manualCTRL
    := drive.bM1switch;
END_TRANSITION
STEP manualCTRL:
    manualCTRL_entry(P1);  // entry action
    manualCTRL_active(N);  // step action
    manualCTRL_exit(P0);  // exit action
END_STEP
TRANSITION FROM manualCTRL TO Init
    := not drive.bM1switch;
END_TRANSITION

ACTION manualCTRL_active:
IF drive.ATV_TPDO_Input1_Status_Word = atv_status.rdy2SwitchON THEN 
	drive.ATV_RPDO_Output1_Control_Word := 7;
END_IF

IF drive.ATV_TPDO_Input1_Status_Word = atv_status.SwitchedON THEN 
	drive.ATV_RPDO_Output1_Control_Word := 15;
	drive.bM1active := TRUE; 
END_IF

drive.bFeedMotor2 := TRUE;
END_ACTION

ACTION manualCTRL_entry:
drive.ATV_RPDO_Output2_Target_Velocity := 1000;
drive.ATV_RPDO_Output1_Control_Word := 6;
END_ACTION

ACTION manualCTRL_exit:
drive.ATV_RPDO_Output1_Control_Word := 7; 
drive.bM1active := FALSE;

drive.bFeedMotor2 := FALSE;
END_ACTION

END_PROGRAM

// ---- POUs/CabinetSwitch.TcPOU
PROGRAM CabinetSwitch
VAR
END_VAR

// Written 08.08.2023 by Daniel Kelly

// Program provides control for the lights inside the switches

drive.bEmergencyLamp1 := NOT drive.bEstop; // turns on the lamp inside the emergency switch
drive.bstartprocessSwitchlamp := drive.bStartProcess OR drive.bShortFeed; // turns on the lamp inside the main switch
drive.bfeedmotorSwitchlamp := drive.bM1switch; // turns on the lamp inside the main feeding motor switch
drive.bremovalmotorSwitchlamp := drive.bM2switch; // turns on the lamp inside removal motor switch
drive.bValveSwitchLamp := drive.ValveSwitch; 
drive.bEmptySystemSwitchLamp := drive.RemovalSwitch;

END_PROGRAM

// ---- POUs/ValveManualControl.TcPOU
PROGRAM ValveManualControl
VAR
END_VAR

// written 18.08.2023 by Daniel Kelly

// Program provides manual control for the valves
// Valve1Open opens the top valve
// Valve1Close closes the top valve
// Valve2Open opens the bottom valve
// Valve2Close closes the bottom valve

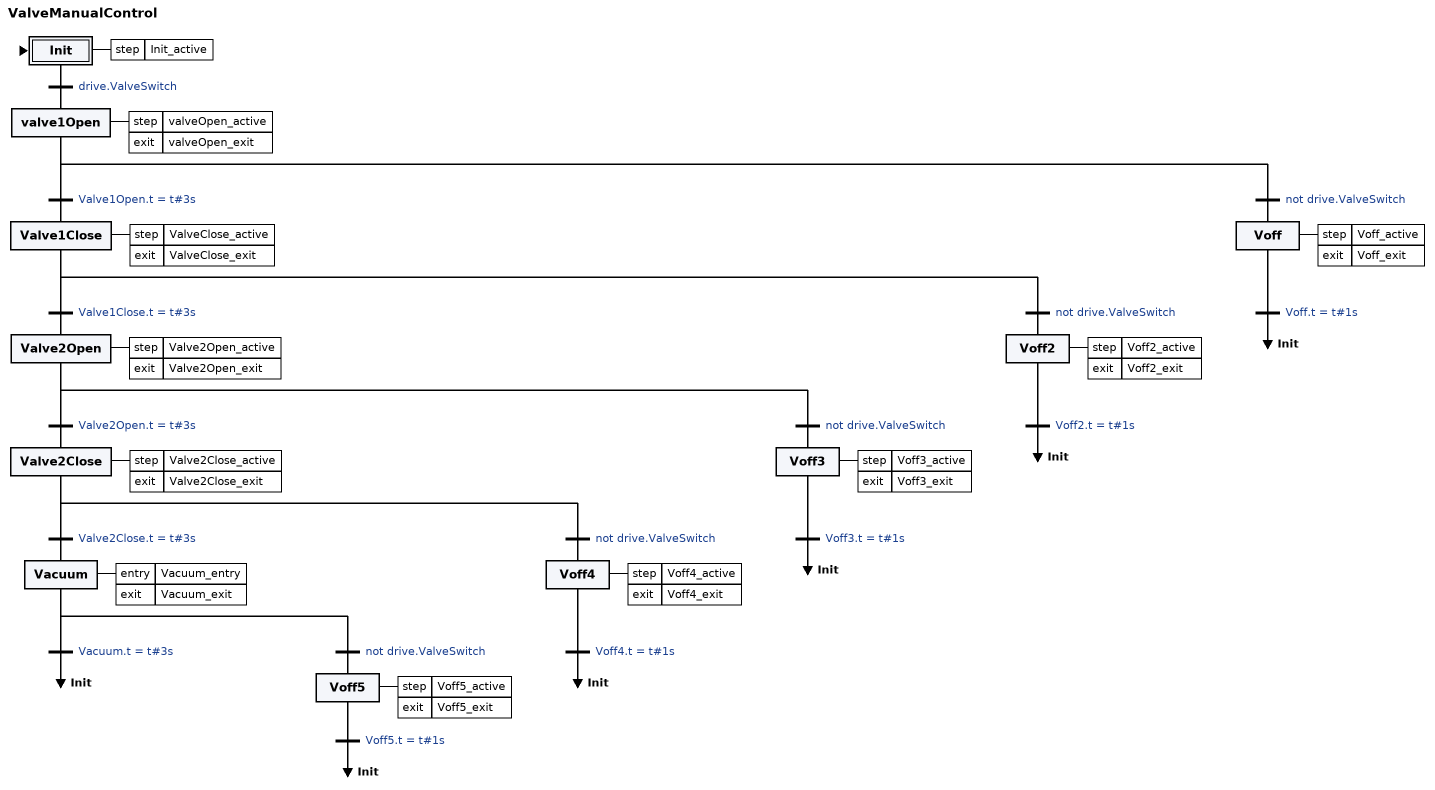
INITIAL_STEP Init:
    Init_active(N);  // step action
END_STEP
TRANSITION FROM Init TO valve1Open
    := drive.ValveSwitch;
END_TRANSITION
STEP valve1Open:
    valveOpen_active(N);  // step action
    valveOpen_exit(P0);  // exit action
END_STEP
TRANSITION FROM valve1Open TO Valve1Close
    := Valve1Open.t = t#3s;
END_TRANSITION
TRANSITION FROM valve1Open TO Voff
    := not drive.ValveSwitch;
END_TRANSITION
STEP Voff:
    Voff_active(N);  // step action
    Voff_exit(P0);  // exit action
END_STEP
TRANSITION FROM Voff TO Init
    := Voff.t = t#1s;
END_TRANSITION
STEP Valve1Close:
    ValveClose_active(N);  // step action
    ValveClose_exit(P0);  // exit action
END_STEP
TRANSITION FROM Valve1Close TO Valve2Open
    := Valve1Close.t = t#3s;
END_TRANSITION
TRANSITION FROM Valve1Close TO Voff2
    := not drive.ValveSwitch;
END_TRANSITION
STEP Voff2:
    Voff2_active(N);  // step action
    Voff2_exit(P0);  // exit action
END_STEP
TRANSITION FROM Voff2 TO Init
    := Voff2.t = t#1s;
END_TRANSITION
STEP Valve2Open:
    Valve2Open_active(N);  // step action
    Valve2Open_exit(P0);  // exit action
END_STEP
TRANSITION FROM Valve2Open TO Valve2Close
    := Valve2Open.t = t#3s;
END_TRANSITION
TRANSITION FROM Valve2Open TO Voff3
    := not drive.ValveSwitch;
END_TRANSITION
STEP Voff3:
    Voff3_active(N);  // step action
    Voff3_exit(P0);  // exit action
END_STEP
TRANSITION FROM Voff3 TO Init
    := Voff3.t = t#1s;
END_TRANSITION
STEP Valve2Close:
    Valve2Close_active(N);  // step action
    Valve2Close_exit(P0);  // exit action
END_STEP
TRANSITION FROM Valve2Close TO Vacuum
    := Valve2Close.t = t#3s;
END_TRANSITION
TRANSITION FROM Valve2Close TO Voff4
    := not drive.ValveSwitch;
END_TRANSITION
STEP Voff4:
    Voff4_active(N);  // step action
    Voff4_exit(P0);  // exit action
END_STEP
TRANSITION FROM Voff4 TO Init
    := Voff4.t = t#1s;
END_TRANSITION
STEP Vacuum:
    Vacuum_entry(P1);  // entry action
    Vacuum_exit(P0);  // exit action
END_STEP
TRANSITION FROM Vacuum TO Init
    := Vacuum.t = t#3s;
END_TRANSITION
TRANSITION FROM Vacuum TO Voff5
    := not drive.ValveSwitch;
END_TRANSITION
STEP Voff5:
    Voff5_active(N);  // step action
    Voff5_exit(P0);  // exit action
END_STEP
TRANSITION FROM Voff5 TO Init
    := Voff5.t = t#1s;
END_TRANSITION

ACTION Init_active:
//drive.LeftSolenoid := FALSE;
//drive.LeftSolenoid2 := FALSE;
//drive.RightSolenoid := FALSE;
//drive.RightSolenoid2 := FALSE;
END_ACTION

ACTION Vacuum_entry:
drive.bVacuum := TRUE;
END_ACTION

ACTION Vacuum_exit:
drive.bVacuum := FALSE;
END_ACTION

ACTION Valve2Close_active:
drive.CloseBottomValve := TRUE;
END_ACTION

ACTION Valve2Close_exit:
drive.CloseBottomValve := FALSE;
drive.bValveLamp := FALSE;
END_ACTION

ACTION Valve2Open_active:
drive.OpenBottomValve := TRUE;
END_ACTION

ACTION Valve2Open_exit:
drive.OpenBottomValve := FALSE;
END_ACTION

ACTION ValveClose_active:
drive.OpenTopValve := FALSE;
drive.CloseTopValve := TRUE;
END_ACTION

ACTION ValveClose_exit:
drive.CloseTopValve := FALSE;
END_ACTION

ACTION valveOpen_active:
drive.OpenTopValve := TRUE;
END_ACTION

ACTION valveOpen_exit:
drive.OpenTopValve := FALSE;
END_ACTION

ACTION Voff_active:
drive.OpenTopValve := FALSE;
drive.CloseTopValve := TRUE;
drive.OpenBottomValve := FALSE;
drive.CloseBottomValve := TRUE;
END_ACTION

ACTION Voff_exit:
drive.CloseBottomValve := FALSE;
drive.CloseTopValve := FALSE;
END_ACTION

ACTION Voff2_active:
drive.OpenTopValve := FALSE;
drive.CloseTopValve := TRUE;
drive.OpenBottomValve := FALSE;
drive.CloseBottomValve := TRUE;
END_ACTION

ACTION Voff2_exit:
drive.CloseBottomValve := FALSE;
drive.CloseTopValve := FALSE;
END_ACTION

ACTION Voff3_active:
drive.OpenTopValve := FALSE;
drive.CloseTopValve := TRUE;
drive.OpenBottomValve := FALSE;
drive.CloseBottomValve := TRUE;
END_ACTION

ACTION Voff3_exit:
drive.CloseBottomValve := FALSE;
drive.CloseTopValve := FALSE;
END_ACTION

ACTION Voff4_active:
drive.OpenTopValve := FALSE;
drive.CloseTopValve := TRUE;
drive.OpenBottomValve := FALSE;
drive.CloseBottomValve := TRUE;
END_ACTION

ACTION Voff4_exit:
drive.CloseBottomValve := FALSE;
drive.CloseTopValve := FALSE;
END_ACTION

ACTION Voff5_active:
drive.OpenTopValve := FALSE;
drive.CloseTopValve := TRUE;
drive.OpenBottomValve := FALSE;
drive.CloseBottomValve := TRUE;
END_ACTION

ACTION Voff5_exit:
drive.CloseBottomValve := FALSE;
drive.CloseTopValve := FALSE;
END_ACTION

END_PROGRAM

// ---- POUs/Scaling.TcPOU
PROGRAM Scaling
VAR
END_VAR
// written 10.07.2023 by Daniel Kelly

// Program provides scaling for the signals from the thermocouples

drive.ScaledThermoCouple1Value := drive.RawThermoCouple1Value * (1000.0/32767); // not in use
drive.ScaledThermoCouple2Value := drive.RawThermoCouple2Value * (1000.0/32767);

END_PROGRAM

// ---- POUs/FeedMotor2Manualcontrol.TcPOU
PROGRAM FeedMotor2Manualcontrol
VAR
END_VAR

// Written 10.08.2023 by Daniel Kelly

// Program provides manual control of the removal motor M2 via its switch

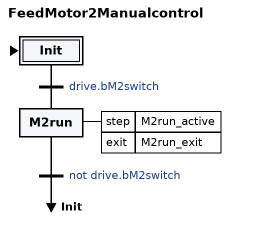
INITIAL_STEP Init:
END_STEP
TRANSITION FROM Init TO M2run
    := drive.bM2switch;
END_TRANSITION
STEP M2run:
    M2run_active(N);  // step action
    M2run_exit(P0);  // exit action
END_STEP
TRANSITION FROM M2run TO Init
    := not drive.bM2switch;
END_TRANSITION

ACTION M2run_active:
drive.bRemovalMotor := TRUE;
END_ACTION

ACTION M2run_exit:
drive.bRemovalMotor := FALSE;
END_ACTION

ACTION manualCTRL2_active:
drive.bRemovalMotor := TRUE; 
drive.bM2active := TRUE;
END_ACTION

ACTION manualCTRL2_entry:
//drive.bRemovalMotor := TRUE; 
//drive.bM2active := TRUE;
END_ACTION

ACTION manualCTRL2_exit:
drive.bRemovalMotor := FALSE; 
drive.bM2active := FALSE;
END_ACTION

END_PROGRAM

// ---- POUs/RemovalProgram.TcPOU
PROGRAM RemovalProgram
VAR
END_VAR

// Written 25.8.2023 by Daniel Kelly

// The purpose of this POU is to automate the emptying of the system
//OpenValves will open both top and bottom valves
//RemovalMotorON will turn on the removal motor
//FM1_ON turns on the grey feeding motor M1
// The steps OFF1, OFF2 etc. turns of the removal motor and both top and bottom valves

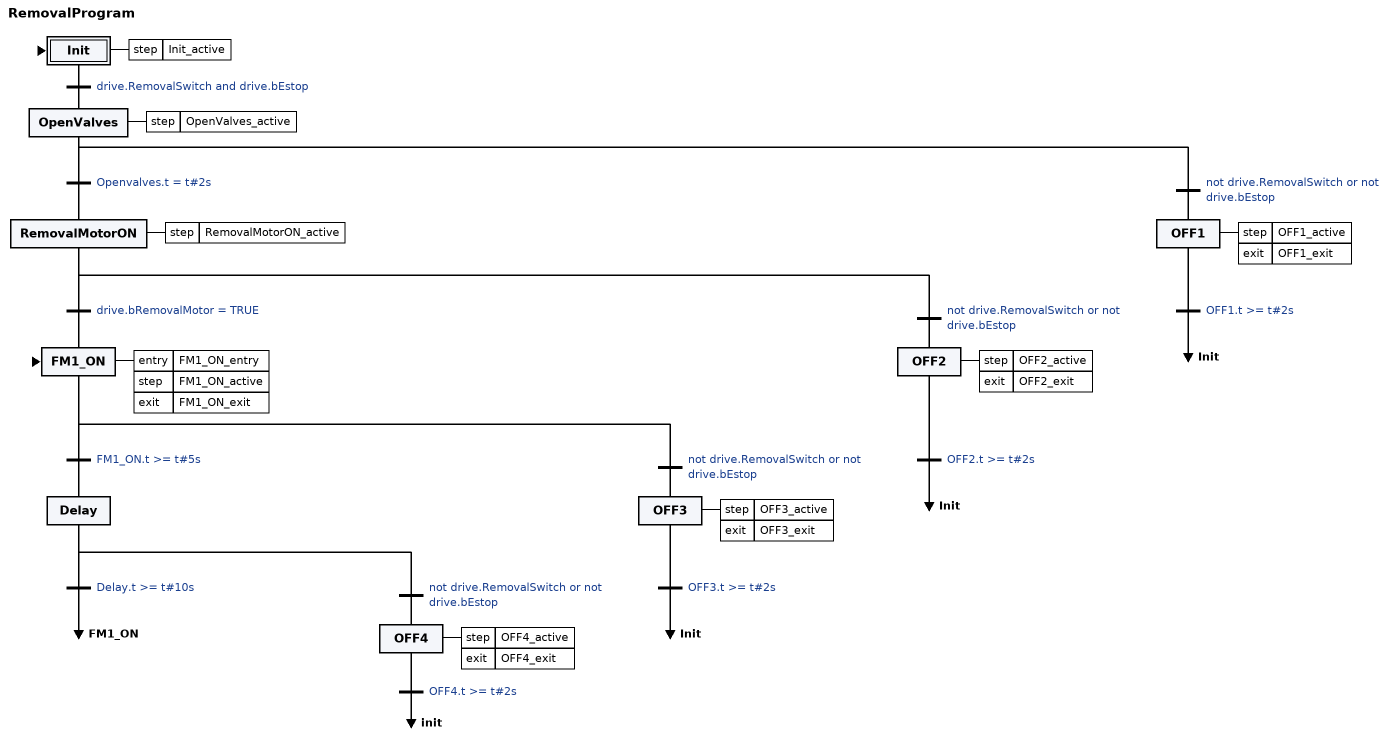
INITIAL_STEP Init:
    Init_active(N);  // step action
END_STEP
TRANSITION FROM Init TO OpenValves
    := drive.RemovalSwitch and drive.bEstop;
END_TRANSITION
STEP OpenValves:
    OpenValves_active(N);  // step action
END_STEP
TRANSITION FROM OpenValves TO RemovalMotorON
    := Openvalves.t = t#2s;
END_TRANSITION
TRANSITION FROM OpenValves TO OFF1
    := not drive.RemovalSwitch or not drive.bEstop;
END_TRANSITION
STEP OFF1:
    OFF1_active(N);  // step action
    OFF1_exit(P0);  // exit action
END_STEP
TRANSITION FROM OFF1 TO Init
    := OFF1.t >= t#2s;
END_TRANSITION
STEP RemovalMotorON:
    RemovalMotorON_active(N);  // step action
END_STEP
TRANSITION FROM RemovalMotorON TO FM1_ON
    := drive.bRemovalMotor = TRUE;
END_TRANSITION
TRANSITION FROM RemovalMotorON TO OFF2
    := not drive.RemovalSwitch or not drive.bEstop;
END_TRANSITION
STEP OFF2:
    OFF2_active(N);  // step action
    OFF2_exit(P0);  // exit action
END_STEP
TRANSITION FROM OFF2 TO Init
    := OFF2.t >= t#2s;
END_TRANSITION
STEP FM1_ON:
    FM1_ON_entry(P1);  // entry action
    FM1_ON_active(N);  // step action
    FM1_ON_exit(P0);  // exit action
END_STEP
TRANSITION FROM FM1_ON TO Delay
    := FM1_ON.t >= t#5s;
END_TRANSITION
TRANSITION FROM FM1_ON TO OFF3
    := not drive.RemovalSwitch or not drive.bEstop;
END_TRANSITION
STEP OFF3:
    OFF3_active(N);  // step action
    OFF3_exit(P0);  // exit action
END_STEP
TRANSITION FROM OFF3 TO Init
    := OFF3.t >= t#2s;
END_TRANSITION
STEP Delay:
END_STEP
TRANSITION FROM Delay TO FM1_ON
    := Delay.t >= t#10s;
END_TRANSITION
TRANSITION FROM Delay TO OFF4
    := not drive.RemovalSwitch or not drive.bEstop;
END_TRANSITION
STEP OFF4:
    OFF4_active(N);  // step action
    OFF4_exit(P0);  // exit action
END_STEP
TRANSITION FROM OFF4 TO init
    := OFF4.t >= t#2s;
END_TRANSITION

ACTION FM1_ON_active:
IF drive.ATV_TPDO_Input1_Status_Word = atv_status.rdy2SwitchON THEN 
	drive.ATV_RPDO_Output1_Control_Word := 7;
END_IF

IF drive.ATV_TPDO_Input1_Status_Word = atv_status.SwitchedON THEN 
	drive.ATV_RPDO_Output1_Control_Word := 15;
	
END_IF

drive.bM1active := TRUE;
END_ACTION

ACTION FM1_ON_entry:
drive.ATV_RPDO_Output2_Target_Velocity := 1000;
drive.ATV_RPDO_Output1_Control_Word := 6;
END_ACTION

ACTION FM1_ON_exit:
drive.ATV_RPDO_Output1_Control_Word := 7; 
drive.bM1active := FALSE;
END_ACTION

ACTION Init_active:

END_ACTION

ACTION OFF1_active:
drive.bRemovalMotor := FALSE;
drive.CloseTopValve := TRUE;
drive.CloseBottomValve := TRUE;

drive.OpenTopValve := FALSE;
drive.OpenBottomValve := FALSE;

drive.bValveLamp := FALSE;
END_ACTION

ACTION OFF1_exit:
drive.CloseBottomValve := FALSE;
drive.CloseTopValve := FALSE;
END_ACTION

ACTION OFF2_active:
drive.bRemovalMotor := FALSE;
drive.CloseTopValve := TRUE;
drive.CloseBottomValve := TRUE;

drive.OpenTopValve := FALSE;
drive.OpenBottomValve := FALSE;

drive.bValveLamp := FALSE;
END_ACTION

ACTION OFF2_exit:
drive.CloseBottomValve := FALSE;
drive.CloseTopValve := FALSE;
END_ACTION

ACTION OFF3_active:
drive.bRemovalMotor := FALSE;
drive.CloseTopValve := TRUE;
drive.CloseBottomValve := TRUE;

drive.OpenTopValve := FALSE;
drive.OpenBottomValve := FALSE;

drive.bValveLamp := FALSE;
drive.bM1active := FALSE;
END_ACTION

ACTION OFF3_exit:
drive.CloseBottomValve := FALSE;
drive.CloseTopValve := FALSE;
END_ACTION

ACTION OFF4_active:
drive.bRemovalMotor := FALSE;
drive.CloseTopValve := TRUE;
drive.CloseBottomValve := TRUE;

drive.OpenTopValve := FALSE;
drive.OpenBottomValve := FALSE;

drive.bValveLamp := false;
END_ACTION

ACTION OFF4_exit:
drive.CloseBottomValve := FALSE;
drive.CloseTopValve := FALSE;
END_ACTION

ACTION OpenValves_active:
drive.CloseTopValve := FALSE;
drive.CloseBottomValve := FALSE;


drive.OpenTopValve := TRUE;
drive.OpenBottomValve := TRUE;

drive.bValveLamp := TRUE;
END_ACTION

ACTION RemovalMotorON_active:
drive.bRemovalMotor := TRUE;
END_ACTION

ACTION TurnOFFValve_active:

END_ACTION

END_PROGRAM

// ---- GlobalTextList.TcGTLO
TEXTLIST GlobalTextList
  733 = ' %d'
  941 = ' %d / 5'
  249 = '%'
  828 = '%.2f  C'
  161 = 'b g'
  106 = 'C'
  558 = 'Feeding motor 1'
  639 = 'Feeding Motor 1'
  177 = 'Feeding motor 2'
  153 = 'Feeding Motor 2'
  972 = 'Feeding motor 3'
  146 = 'Number of cycles before product release'
  744 = 'Process Active'
  554 = 'removal motor'
  562 = 'Removal motor'
  707 = 'Removal Motor'
  391 = 'Valves'
END_TEXTLIST

// ---- VISUs/Visualization.TcVIS
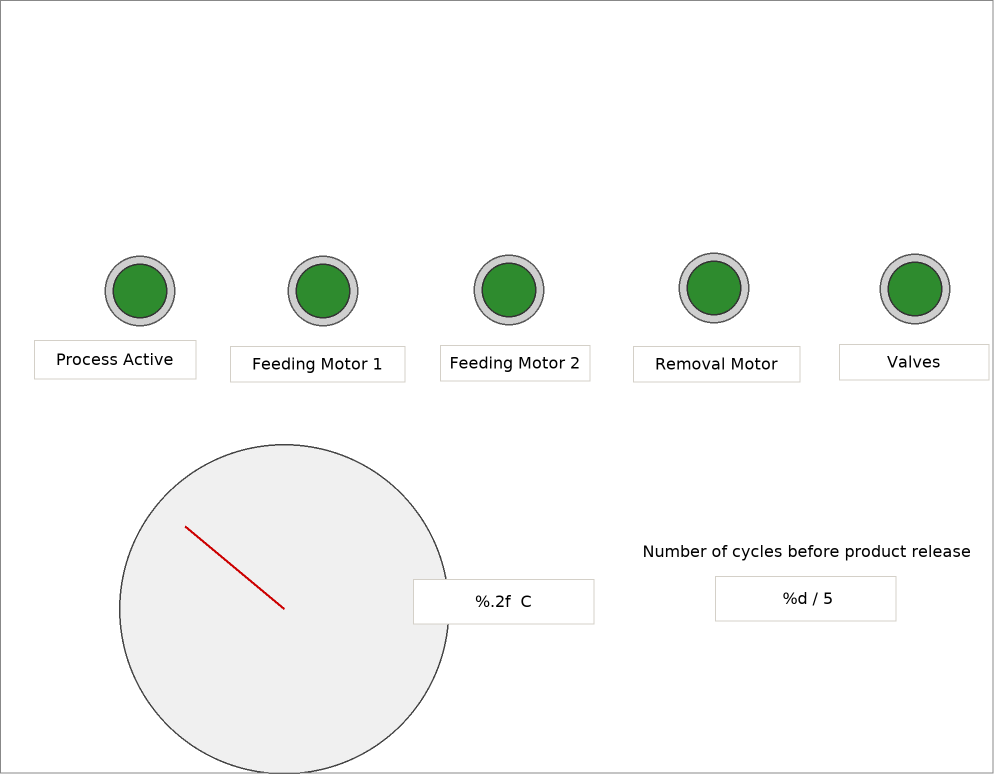
VISUALIZATION Visualization  // 994x774, background image ImagePool.Keskisuuri+600px(näytöille,+RGB,+JPG)+HAMK_HAMK_Logo_text_large_FIN
    Textfield (34,340 162x39), "Process Active"
    Lamp1 (97,250 86x82), variable: drive.bProcessActive, style: Lamp-Lamp1-Green
    Lamp1 (280,250 86x82), variable: drive.bM1active, style: Lamp-Lamp1-Green
    Lamp1 (466,249 86x82), variable: drive.bFeedMotor2Lamp, style: Lamp-Lamp1-Green
    Lamp1 (671,247 86x82), variable: drive.bM2active, style: Lamp-Lamp1-Green
    Textfield (230,346 175x36), "Feeding Motor 1"
    Textfield (440,345 150x36), "Feeding Motor 2"
    Textfield (633,346 167x36), "Removal Motor"
    Meter360 (33,444 502x330), value: drive.ScaledThermoCouple2Value, style: Meter-Meter360-Yellow, scale format: %.1f, scale 0..800
    Lamp1 (872,248 86x82), variable: drive.bValveLamp, style: Lamp-Lamp1-Green
    Textfield (839,344 150x36), "Valves"
    Textfield (413,579 181x45), "%.2f C", text variable: drive.ScaledThermoCouple2Value
    Textfield (715,576 181x45), "%d / 5", text variable: drive.itopvalvecount
    Label (620,519 374x65), "Number of cycles before product release"
END_VISUALIZATION
